FUNCTION_BLOCK LOG_16 (* Ring Logger for ANY Datattype. *)
  (* Standard: 61499-2 *)
  (* Version 1.0, 2025-10-18, Franz Höpfinger, initial API and implementation and/or initial documentation *)
  PACKAGE logiBUS::utils::logging;
  {SET_ATTRIBUTE(eclipse4diac::core::GenericClassName, 'GEN_LOG')}
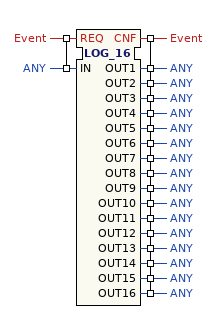
  EVENT_INPUT
    REQ WITH IN; (* Service Request *)
  END_EVENT
  EVENT_OUTPUT
    CNF WITH OUT1, OUT2, OUT3, OUT4, OUT5, OUT6, OUT7, OUT8, OUT9, OUT10, OUT11, OUT12, OUT13, OUT14, OUT15, OUT16; (* Confirmation of Requested Service *)
  END_EVENT
  VAR_INPUT
    IN : ANY;
  END_VAR
  VAR_OUTPUT
    OUT1 : ANY;
    OUT2 : ANY;
    OUT3 : ANY;
    OUT4 : ANY;
    OUT5 : ANY;
    OUT6 : ANY;
    OUT7 : ANY;
    OUT8 : ANY;
    OUT9 : ANY;
    OUT10 : ANY;
    OUT11 : ANY;
    OUT12 : ANY;
    OUT13 : ANY;
    OUT14 : ANY;
    OUT15 : ANY;
    OUT16 : ANY;
  END_VAR
END_FUNCTION_BLOCK
